{attribute 'strict'}
TYPE MainState_enum :
(
	MS_DISABLED					:= 0,
	MS_INITIALIZING_MOVERS		:= 10,
	MS_ENABLING_MOVERS			:= 20,
	MS_INITIALIZING_OBJECTIVES	:= 30,
	MS_ENABLED					:= 40,
	MS_RUN						:= 50,
	MS_STOPPING					:= 60,
	MS_DISABLING				:= 70,
	MS_ERROR					:= 80,
	MS_STOPPED					:= 90,
	MS_DEBUG					:= 1000
);
END_TYPE

(* stored: Version 1.1.0.1, ProductVersion 3.1.4024.11
   DUT MainState_enum: Id {62255fa4-5620-44dc-b5d1-8a2be4061452} *)
